(* PLC project Generated.project, CODESYS CODESYS V3.5 SP19 Patch 1 *)
(* stored: creationDateTime 2026-09-06T13:00:42.441732, modificationDateTime 2026-09-06T13:00:42.441732 *)

(* ======================================================================= 📊 ST_fbWinchLoadEstimator_Table — Table empirique de charge estimée ─────────────────────────────────────────────────────────────── 🎯 Rôle : Matrice 5x5 d'estimation de charge (palier commandé x bande vitesse) 📄 Doc métier : DOC/AF/AF_Partie-10_Fonction_Winch_v2.1.md ======================================================================= *)
TYPE ST_fbWinchLoadEstimator_Table : STRUCT
  IsConfigured : BOOL;  (* Validation explicite de la table *)
  LoadPctByStepAndSpeedBand : ARRAY[1..5] OF ARRAY[1..5] OF REAL;  (* Matrice [palier][bande_vitesse] charge (%) *)
END_STRUCT;
END_TYPE
